// TIA Portal V20 export
TYPE "LConSMC_typeSectionalDriveInput"
// stored: Access Published
   STRUCT
      enable : Bool := FALSE;   // TRUE: Freigabe des Bausteins. Mit steigender Flanke erfolgt Parametervalidierung und Kommunikation mit dem Antrieb FALSE: Baustein ausschalten / TRUE: Enable function block. WIth rising edge a validation of parameter is done and communication with drive is started FALSE: Disable the function block
      speedMatch : Bool;   // TRUE: Freigabe der Bahngeschwindigkeitssolwert ("lineAxisMotionVector"). Der Antrieb synchronisiert auf die Bahngeschwindigkeit auf mit Hilfe der Synchronisationsdynamiken. Ist der Antrieb synchron so wird der Ausgang "inSync" = TRUE. FALSE: Der Antrieb verzögert bis zum Stillstand mit Hilfe der Stoppdynamiken / True: Enable web velocity setpoint ("lineAxisMotionVector"). The drive will synchronize up to web velocity using syncronization dynamics. If the velocity is reached the output "inSync" will become TRUE. FALSE: Drive will decelerate to standstill using stop dynamics
      CntrlEnable : Bool := FALSE;   // TRUE: Freigabe der Bahnzugregelung (Freigabe Drehmomentengrenzen/ Tänzersollwert etc.) / TRUE: Enable web tension control (enable torque limits, dancer position setpoint etc.)
      jogPos : Bool := FALSE;   // TRUE: Antrieb wird in positive Richtung vertippt (siehe config.dynamics.jogDynamics) / TRUE: Drive is jogged in positive direction (see config.dynamics.jogDynamics)
      jogNeg : Bool := FALSE;   // TRUE: Antrieb wird in negative Richtung vertippt (siehe config.dynamics.jogDynamics) / TRUE: Drive is jogged in negative direction (see config.dynamics.jogDynamics)
      lineAxisMotionVector : "LConSMC_typeMotionVector";   // Sollwert der Bahn (Position/Geschwindigkeit/Beschleunigung) / Setpoint of the web (position/velocity/acceleration)
      additionalVelocity : LReal := 0.0;   // [m/min] / [ft/min] Zusätzliche Bahngeschwindigkeit (immer aktiv) / [m/min] / [ft/min] Additional web velocity (always enabled)
      draw : LReal := 1.0;   // Draw Faktor für den Regelungsmodus 4 (DRAW_CONTROL). Sollwert = Bahnsollwert * draw / Draw factor for control mode 4 (DRAW CONTROL). Velocity setpoint = webVelocity * draw
      typeOfDrive : Int := 0;   // Definition der Bahnzugrichtung 0: Bahnzug vor der Rolle wird geregelt (Pull) 1: Bahnzug nach der Rolle wird geregelt (Push) / Definition of web tension direction 0: Web tension bevor the roll is controlled (Pull) 1: Web tension after the roll is controlled (Push)
      controlMode : Int := 0;   // Regelungsmodus 0:Tänzerlageregelung via Drehzahladaption 1: Zugmessdose via Drehzahladaption 2: Zugmessdose via Drehmomentenadaption 3: Indirekte Zugregelung 4: Geschwindigkeitsrelation (Draw) / Tension control mode 0: Dancer via speed setpoint adaption 1: Load cell via speed setpoint adaption 2: Load cell via torque limits 3: Indirect tension control 4: Speed setpoint relation (Draw) 5: Indirect tension control vis speed setpoint adaption
      CntrlSetpoint : LReal := 0.0;   // Zugsollwert [N]/[Lbf] / Lagesollwert Tänzer [%] / Tension setpoint [N]/[Lbf] / Dancer position setpoint [%]
      CntrlActual : LReal := 0.0;   // Istzug[N]/[Lbf] / Lageistwert Tänzer [%] / Tension actual value [N]/[Lbf] / Dancer actual position [%]
      tCycle : Real := 0.0;   // [ms] Zykluszeit in der der Baustein aufgerufen wird / [ms] Cycle time the function block is called
      axis : DB_ANY;   // Bahnzugachse / Sectional drive axis
   END_STRUCT;
END_TYPE
